(*
    Verifies that the function IS_TEST_FINISHED('Name') works as intended.
*)
FUNCTION_BLOCK FB_CheckIfSpecificTestIsFinished EXTENDS TcUnit.FB_TestSuite

CheckBeforeAndAfterFinishing();

METHOD CheckBeforeAndAfterFinishing
TEST('CheckBeforeAndAfterFinishing');

AssertEquals_BOOL(Expected := FALSE,
                  Actual := IS_TEST_FINISHED('CheckBeforeAndAfterFinishing'),
                  Message:='Values differ before finishing');

TEST_FINISHED();

AssertEquals_BOOL(Expected := TRUE,
                  Actual := IS_TEST_FINISHED('CheckBeforeAndAfterFinishing'),
                  Message:='Values differ after finishing');
END_METHOD

END_FUNCTION_BLOCK

(* stored: Version 1.1.0.1, ProductVersion 3.1.4022.18
   POU FB_CheckIfSpecificTestIsFinished: Id {2acea95d-ab41-4d72-9612-66cd6d5b13cc}, SpecialFunc None
   Method CheckBeforeAndAfterFinishing: Id {bc4e3608-724f-4d4e-ad3f-c0950dd8383e} *)
